TYPE ST_TEST_AnyBuffer_Element :
STRUCT
	id				: INT;
	name			: STRING;
END_STRUCT
END_TYPE

(* stored: Version 1.1.0.1, ProductVersion 3.1.4026.18
   DUT ST_TEST_AnyBuffer_Element: Id {e3dc4dcc-488f-4f5f-a42c-7a4d013e23a8} *)
